FUNCTION_BLOCK CentralizedController (* Basic Function Block Type *)
  (* Standard: 61499-2 *)
  (* Version 0.0, 2/16/2024, midxav, Template *)
  PACKAGE Main;
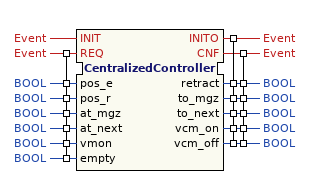
  EVENT_INPUT
    INIT; (* Initialization Request *)
    REQ WITH pos_e, pos_r, at_mgz, at_next, vmon, empty; (* Normal Execution Request *)
  END_EVENT
  EVENT_OUTPUT
    INITO WITH retract, to_mgz, to_next, vcm_on, vcm_off; (* Initialization Confirm *)
    CNF WITH retract, to_mgz, to_next, vcm_on, vcm_off; (* Execution Confirmation *)
  END_EVENT
  VAR_INPUT
    pos_e : BOOL; (* Input event qualifier *)
    pos_r : BOOL;
    at_mgz : BOOL;
    at_next : BOOL;
    vmon : BOOL;
    empty : BOOL;
  END_VAR
  VAR_OUTPUT
    retract : BOOL; (* Output event qualifier *)
    to_mgz : BOOL;
    to_next : BOOL;
    vcm_on : BOOL;
    vcm_off : BOOL;
  END_VAR
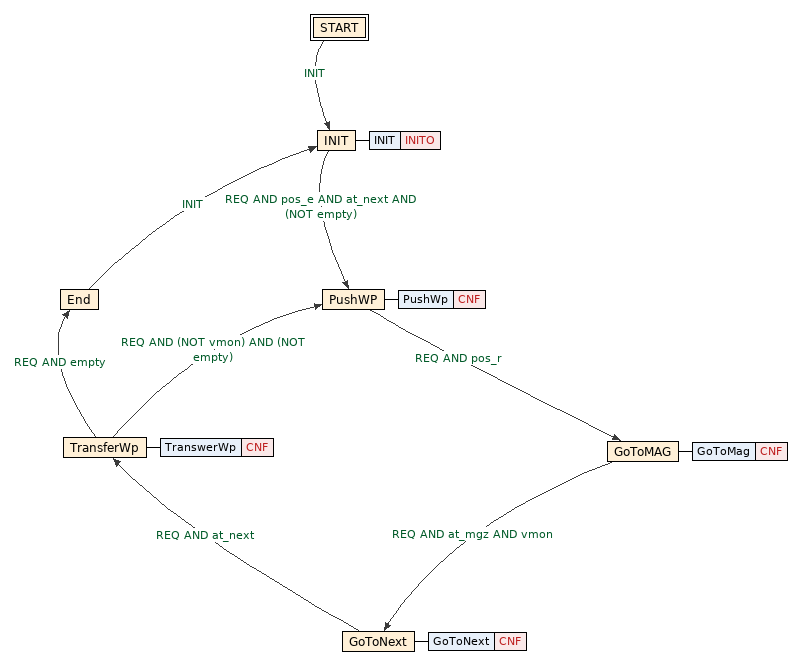
  EC_STATES
    START; (* Initial State *)
    INIT : INIT -> INITO; (* Initialization *)
    GoToMAG : GoToMag -> CNF;
    PushWP : PushWp -> CNF;
    GoToNext : GoToNext -> CNF;
    TransferWp : TranswerWp -> CNF;
    End;
  END_STATES
  EC_TRANSITIONS
    START TO INIT := INIT;
    INIT TO PushWP := REQ AND pos_e AND at_next AND (NOT empty);
    PushWP TO GoToMAG := REQ AND pos_r;
    GoToMAG TO GoToNext := REQ AND at_mgz AND vmon;
    TransferWp TO PushWP := REQ AND (NOT vmon) AND (NOT empty);
    GoToNext TO TransferWp := REQ AND at_next;
    TransferWp TO End := REQ AND empty;
    End TO INIT := INIT;
  END_TRANSITIONS
  ALGORITHM INIT IN ST: (* Initialization algorithm *)
retract := FALSE;
to_mgz :=FALSE;
to_next :=TRUE;
vcm_on := FALSE;
vcm_off := TRUE;
  END_ALGORITHM
  ALGORITHM PushWp IN ST:
retract := TRUE;
  END_ALGORITHM
  ALGORITHM GoToMag IN ST:
retract :=FALSE;
to_mgz := TRUE;
to_next := FALSE;
vcm_on := TRUE;
vcm_off := FALSE;
  END_ALGORITHM
  ALGORITHM GoToNext IN ST:
to_mgz := FALSE;
to_next := TRUE;
  END_ALGORITHM
  ALGORITHM TranswerWp IN ST:
vcm_on := FALSE;
vcm_off := TRUE;
  END_ALGORITHM
END_FUNCTION_BLOCK
